// TIA Portal V21 export
TYPE "LBC_typeAxisControlNode"
TITLE = LBC_typeAxisControlNode
// Module related control node wrapper
   STRUCT
      commandConfiguration { ExternalAccessible := 'False'; ExternalVisible := 'False'; ExternalWritable := 'False'} : "LAxisCtrl_typeAxisConfig";
      commands { ExternalAccessible := 'False'; ExternalVisible := 'False'; ExternalWritable := 'False'} : "LBC_typeAxisControlNodeCommands";   // Module related configuration parameters
      monitoring { ExternalAccessible := 'False'; ExternalVisible := 'False'; ExternalWritable := 'False'} : "LBC_typeAxisControlNodeMonitoring";   // Module interface for external systems
   END_STRUCT;
END_TYPE
